Fanuc KAREL source: ko00130.KL

-- PROVISIONAL review KL for V940-1; original PC SHA256 cc30d7e5ebfb189cbe26c1282aec16a3282ccfaf1857c33f03fa0bf4e55b5ae2
-- Incomplete behavior may be omitted. Consult companion uncertainty JSON. Do not deploy.
PROGRAM KO00130
%NOLOCKGROUP
VAR
  R : REAL
  N : REAL
-- UNRESOLVED_DECL CFG type=00001c
-- UNRESOLVED_DECL OUT type=000102
BEGIN
  -- V9_ZERO_TABLE_METADATA_HINT layout=0001; no indexed target words; source/name/runtime held
  -- UNRESOLVED_PC offsets 5-13; opcodes 9D,64,23
  -- UNRESOLVED_PC offsets 18-29; opcodes 2E,23
  -- UNRESOLVED_PC offsets 34-44; opcodes 9D,22,A5
  -- UNRESOLVED_PC offsets 49-106; opcodes 27,22,22,22,22,22,22,22,76,7E,4A
  -- UNRESOLVED_PC offsets 111-115; opcodes 7F
END KO00130
